// TIA Portal V16 export
// export: Created 2021-05-25T16:14:27.0940417Z, ExportSetting WithDefaults, DisplayName Totally Integrated Automation Portal, DisplayVersion V16, DisplayName TIA Portal Version Control Interface, DisplayVersion V16, DisplayName TIA Portal Openness, DisplayVersion V16, DisplayName STEP 7 Professional, DisplayVersion V16, DisplayName STEP 7 Safety, DisplayVersion V16, DisplayName WinCC Unified SCADA Engineering System, DisplayVersion V16
FUNCTION "cmFindStrgEQ" : Bool   // FC220, LAD
{ S7_Optimized_Access := 'TRUE' }
VERSION : 0.1
// stored: AutoNumber false, IsIECCheckEnabled false, SetENOAutomatically false, UDAEnableTagReadback false
   VAR_INPUT
      String1 : String;
      String2 : String;
   END_VAR
BEGIN

REGION Network 1
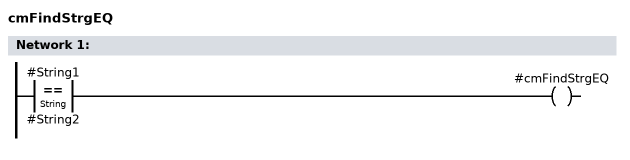
   RUNG wire#powerrail
      { S7_Templates := "SrcType := String" } EQ_Contact(in1 := #String1, in2 := #String2)
      Coil( #cmFindStrgEQ )
   END_RUNG
   // the same network as SCL:
   #cmFindStrgEQ := #String1 = #String2;
END_REGION
END_FUNCTION
